FUNCTION_BLOCK FB_TwoWayPneumaticDrive IMPLEMENTS ITwoPointMovement
VAR_INPUT
END_VAR
VAR_OUTPUT
END_VAR
VAR
END_VAR

{warning 'Eigenschaftenimplementierung hinzufügen'}
PROPERTY InHomePos : BOOL
GET
END_GET
END_PROPERTY

{warning 'Eigenschaftenimplementierung hinzufügen'}
PROPERTY InWorkPos : BOOL
GET
END_GET
END_PROPERTY

{warning 'Methodenimplementierung hinzufügen'}
METHOD ToHomePos : BOOL
END_METHOD

{warning 'Methodenimplementierung hinzufügen'}
METHOD ToWorkPos : BOOL
END_METHOD

END_FUNCTION_BLOCK

(* stored: Version 1.1.0.1, ProductVersion 3.1.4024.11
   POU FB_TwoWayPneumaticDrive: Id {562480a2-ed3c-4fec-9181-18f328b0d4f3}, SpecialFunc None
   Property InHomePos: Id {482e9a7e-cb1b-44e4-a114-a8f7718bcddd}
   Get Get: Id {888bc154-b487-4f7a-b3cd-ec4b7b1a69a4}
   Property InWorkPos: Id {988e3956-3fa1-4176-a942-3692063c2677}
   Get Get: Id {2ae0acd4-d6f6-4e40-a652-b417d095b424}
   Method ToHomePos: Id {06e7a8df-40bc-47df-9d32-40d79090baac}
   Method ToWorkPos: Id {1917dd37-a1b4-4775-8b5b-7503cb460da5} *)
